PROGRAM MAIN
VAR
END_VAR

Aanwezigheids_lichten();
Beamer_Projectorscherm();
SendCommands();

END_PROGRAM

(* stored: Version 1.1.0.1, ProductVersion 3.1.4022.9
   POU MAIN: Id {6a06684d-bcf5-416c-bb0a-1c04413e8cd7}, SpecialFunc None *)
